FUNCTION_BLOCK DigitalInput_Combiner
VAR_GENERIC CONSTANT
	NumberOfCombinedInputs : DINT := 2;
END_VAR
EXTENDS Component IMPLEMENTS I_DigitalInput
VAR
	Inputs : ARRAY[0..(NumberOfCombinedInputs - 1)] OF I_DigitalInput;
	{attribute 'hide'}
	_Force : E_ForceState;
END_VAR

METHOD AddInput
VAR_INPUT
	Input : I_DigitalInput;
END_VAR

VAR
	i : DINT;
END_VAR
FOR i := 0 TO (NumberOfCombinedInputs - 1) DO
	IF Inputs[i] = Input THEN
		RETURN;
	END_IF
END_FOR

FOR i := 0 TO (NumberOfCombinedInputs - 1) DO
	IF Inputs[i] = 0 THEN
		Inputs[i] := Input;
		RETURN;
	END_IF
END_FOR
END_METHOD

{attribute 'monitoring' := 'call'}
PROPERTY Force : E_ForceState
GET
Force := _Force;
END_GET
SET
VAR
	i : DINT;
END_VAR
_Force := Force;
IF Inputs[0] = 0 THEN
	RETURN;
END_IF

FOR i := 0 TO (NumberOfCombinedInputs - 1) DO
	IF Inputs[i] = 0 THEN
		RETURN;
	END_IF

	Inputs[i].Force := Force;
END_FOR
END_SET
END_PROPERTY

{attribute 'monitoring' := 'call'}
PROPERTY IsActive : BOOL
GET
VAR
	i : DINT;
END_VAR
IF Inputs[0] = 0 THEN
	RETURN;
END_IF

IsActive := TRUE;
FOR i := 0 TO (NumberOfCombinedInputs - 1) DO
	IF Inputs[i] = 0 THEN
		RETURN;
	END_IF

	IsActive := IsActive AND Inputs[i].IsActive;
END_FOR
END_GET
END_PROPERTY

END_FUNCTION_BLOCK

(* stored: Version 1.1.0.1, ProductVersion 3.1.4026.18
   POU DigitalInput_Combiner: Id {85b8aac0-ef90-4788-a252-266e964e17ce}, SpecialFunc None
   Method AddInput: Id {bc488cb0-624c-427e-9b71-f3f4aa667e0e}
   Property Force: Id {d2b94b84-9d59-49ca-87c7-768419c63204}
   Get Get: Id {d809e4ed-4465-4d67-836a-9d4973387873}
   Set Set: Id {72f5db18-fb88-4ced-89bc-9eccce7e0b99}
   Property IsActive: Id {8e2bc024-93dc-4f73-8d35-c19f30c0746f}
   Get Get: Id {7286a73a-a3cc-49e6-ba19-38b5212d4306} *)
